// TIA Portal V17 program export: 1 tag tables, 0 data types, 1 data blocks, 2 code blocks (in call order from the OBs), 5 instance data blocks

VAR_GLOBAL   // PLC tag table "Default tag table"
END_VAR

DATA_BLOCK "IO"   // DB1
{ S7_Optimized_Access := 'TRUE' }
VERSION : 0.1
// stored: AutoNumber true, IsOnlyStoredInLoadMemory false, IsRetainMemResEnabled false, IsWriteProtectedInAS false, MemoryReserve 100
   VAR
      start : Bool;
      stop : Bool := true;
      awaryjeOproznianie : Bool := true;
      czasParzenia : Time := T#5S;
      zadanaIloscWody : Real := 500.0;
      zadanaIloscHerbaty : Real := 15.0;
      temperatura : Int;
      przenosnikM1 : Bool;
      mieszalnikM2 : Bool;
      podgrzewaczG1 : Bool;
      otworzZaworZ1 : Bool;
      otworzZasuweZ2 : Bool;
      otworzZasuweZ3 : Bool;
      wodaPoziom : Real;
      lisciePoziom : Real;
      glownyPoziom : Real;
   END_VAR
BEGIN
END_DATA_BLOCK

ORGANIZATION_BLOCK "Main"   // OB1, LAD, ProgramCycle
TITLE = "Main Program Sweep (Cycle)"
{ S7_Optimized_Access := 'TRUE' }
VERSION : 0.1
// stored: AutoNumber true, IsIECCheckEnabled false, SetENOAutomatically false
   VAR_INPUT
      Initial_Call : Bool;   // Initial call of this OB
      Remanence : Bool;   // =True, if remanent data are available
   END_VAR
BEGIN

REGION Network 1: Zadanie finałowe kategorii EKSPERT
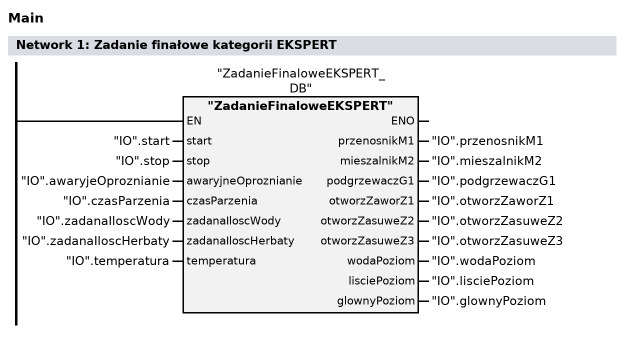
   RUNG wire#powerrail
      "ZadanieFinaloweEKSPERT_DB"(start := "IO".start, stop := "IO".stop, awaryjneOproznianie := "IO".awaryjeOproznianie, czasParzenia := "IO".czasParzenia, zadanaIloscWody := "IO".zadanaIloscWody, zadanaIloscHerbaty := "IO".zadanaIloscHerbaty, temperatura := "IO".temperatura, przenosnikM1 => "IO".przenosnikM1, mieszalnikM2 => "IO".mieszalnikM2, podgrzewaczG1 => "IO".podgrzewaczG1, otworzZaworZ1 => "IO".otworzZaworZ1, otworzZasuweZ2 => "IO".otworzZasuweZ2, otworzZasuweZ3 => "IO".otworzZasuweZ3, wodaPoziom => "IO".wodaPoziom, lisciePoziom => "IO".lisciePoziom, glownyPoziom => "IO".glownyPoziom)
   END_RUNG
   // the same network as SCL:
   "ZadanieFinaloweEKSPERT_DB"(start := "IO".start,   // "ZadanieFinaloweEKSPERT"
                           stop := "IO".stop,
                           awaryjneOproznianie := "IO".awaryjeOproznianie,
                           czasParzenia := "IO".czasParzenia,
                           zadanaIloscWody := "IO".zadanaIloscWody,
                           zadanaIloscHerbaty := "IO".zadanaIloscHerbaty,
                           temperatura := "IO".temperatura,
                           przenosnikM1 => "IO".przenosnikM1,
                           mieszalnikM2 => "IO".mieszalnikM2,
                           podgrzewaczG1 => "IO".podgrzewaczG1,
                           otworzZaworZ1 => "IO".otworzZaworZ1,
                           otworzZasuweZ2 => "IO".otworzZasuweZ2,
                           otworzZasuweZ3 => "IO".otworzZasuweZ3,
                           wodaPoziom => "IO".wodaPoziom,
                           lisciePoziom => "IO".lisciePoziom,
                           glownyPoziom => "IO".glownyPoziom);
END_REGION
END_ORGANIZATION_BLOCK

FUNCTION_BLOCK "ZadanieFinaloweEKSPERT"   // FB1, LAD
TITLE = Zadanie finałowe kategorii EKSPERT
{ S7_Optimized_Access := 'TRUE' }
VERSION : 0.1
// stored: AutoNumber true, IsIECCheckEnabled false, IsRetainMemResEnabled false, MemoryReserve 100, SetENOAutomatically false, UDAEnableTagReadback false
   VAR_INPUT
      start : Bool;
      stop : Bool;
      awaryjneOproznianie : Bool;
      czasParzenia : Time;
      zadanaIloscWody : Real;
      zadanaIloscHerbaty : Real;
      temperatura : Int;
   END_VAR
   VAR_OUTPUT
      przenosnikM1 : Bool;
      mieszalnikM2 : Bool;
      podgrzewaczG1 : Bool;
      otworzZaworZ1 : Bool;
      otworzZasuweZ2 : Bool;
      otworzZasuweZ3 : Bool;
      wodaPoziom : Real := 10000.0;
      lisciePoziom : Real := 100.0;
      glownyPoziom : Real;
   END_VAR
   VAR
      S1 : Bool;
      S2 : Bool;
      S3 : Bool;
      S4 : Bool;
      S5 : Bool;
      S0 : Bool;
      start_edge : Bool;
      stop_edge : Bool;
      awaryjne_edge : Bool;
      S1_Clock : Bool;
      w_glownym_wody : Real;
      w_glownym_herbaty : Real;
      S3_clock : Bool;
      M2_edge : Bool;
      S5_clock : Bool;
   END_VAR
   VAR_TEMP
      temp_norm : Real;
      tempC : Real;
   END_VAR
   VAR_TEMP   // added for the SCL form of the ladder/FBD networks
      _w1 : Bool;
      _w2 : Bool;
      _w3 : Bool;
   END_VAR
BEGIN

REGION Network 1
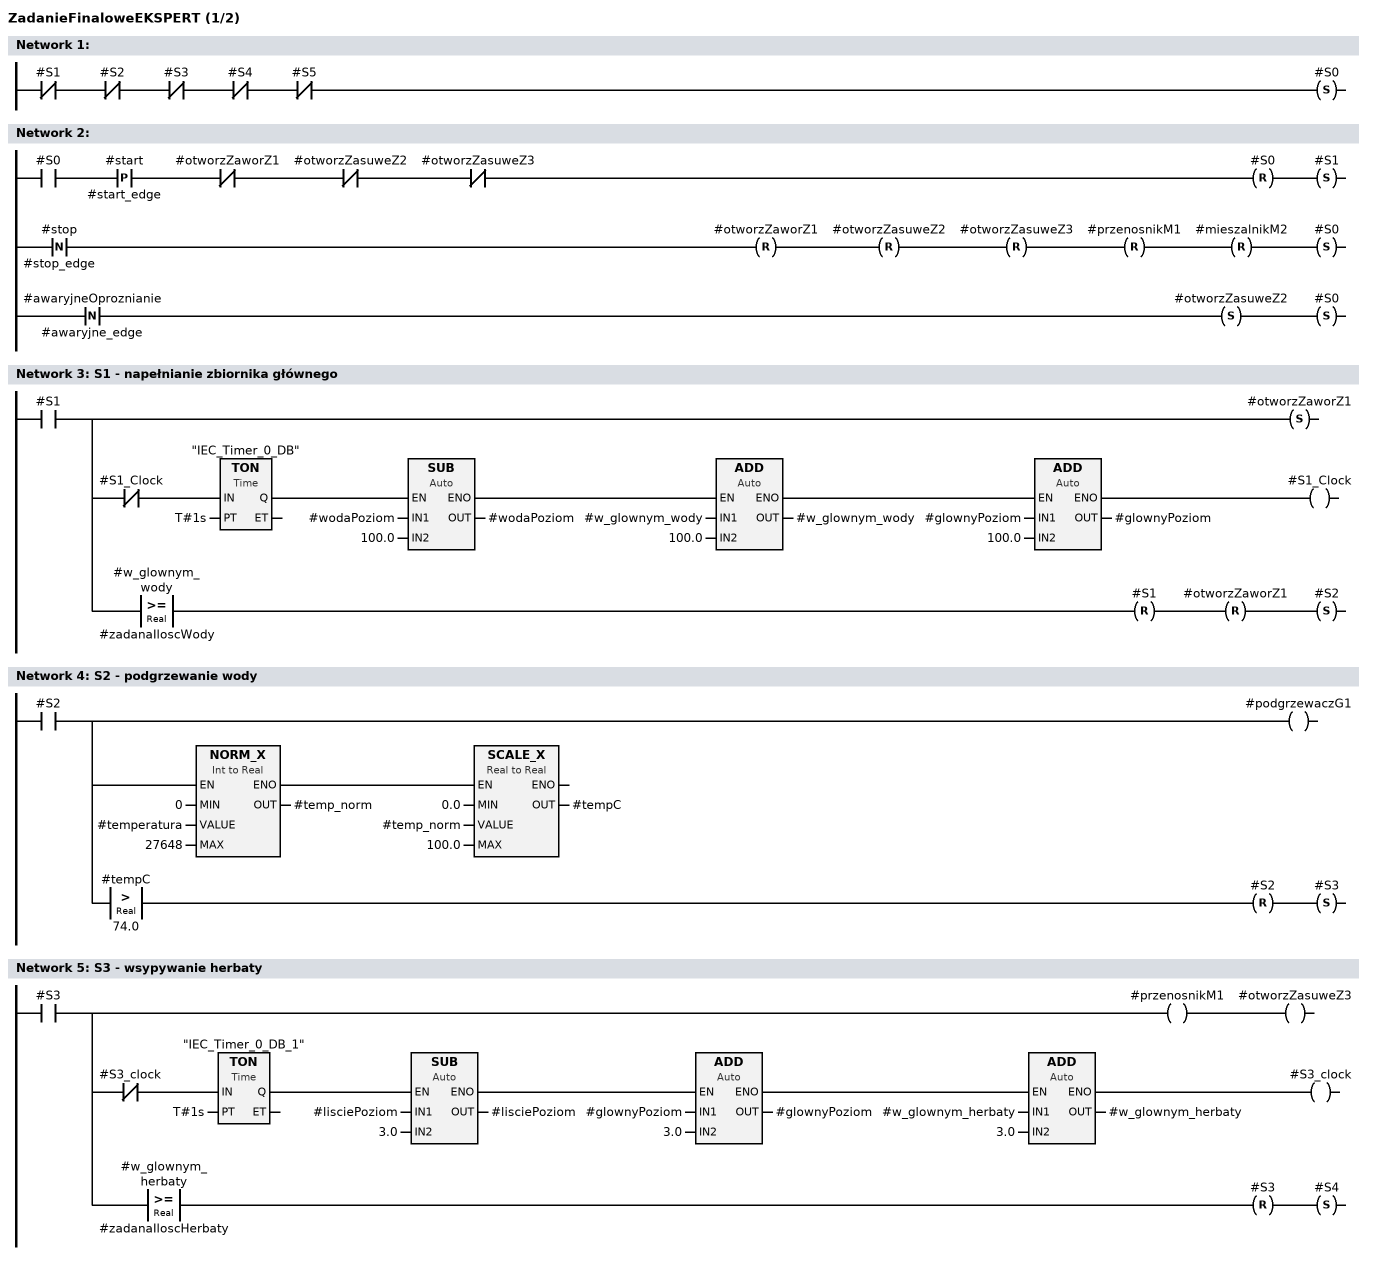
   RUNG wire#powerrail
      I_Contact( #S1 )
      I_Contact( #S2 )
      I_Contact( #S3 )
      I_Contact( #S4 )
      I_Contact( #S5 )
      S_Coil( #S0 )
   END_RUNG
   // the same network as SCL:
   IF NOT #S1 AND NOT #S2 AND NOT #S3 AND NOT #S4 AND NOT #S5 THEN #S0 := TRUE; END_IF;
END_REGION

REGION Network 2
   RUNG wire#powerrail
      Contact( #S0 )
      P_Contact(operand := #start, bit := #start_edge)
      I_Contact( #otworzZaworZ1 )
      I_Contact( #otworzZasuweZ2 )
      I_Contact( #otworzZasuweZ3 )
      R_Coil( #S0 )
      S_Coil( #S1 )
   END_RUNG
   RUNG wire#powerrail
      N_Contact(operand := #stop, bit := #stop_edge)
      R_Coil( #otworzZaworZ1 )
      R_Coil( #otworzZasuweZ2 )
      R_Coil( #otworzZasuweZ3 )
      R_Coil( #przenosnikM1 )
      R_Coil( #mieszalnikM2 )
      S_Coil( #S0 )
   END_RUNG
   RUNG wire#powerrail
      N_Contact(operand := #awaryjneOproznianie, bit := #awaryjne_edge)
      S_Coil( #otworzZasuweZ2 )
      S_Coil( #S0 )
   END_RUNG
   // the same network as SCL:
   #_w1 := #S0 AND #start AND NOT #start_edge;   // rising edge of #start
   #start_edge := #start;
   IF #_w1 AND NOT #otworzZaworZ1 AND NOT #otworzZasuweZ2 AND NOT #otworzZasuweZ3 THEN
       #S0 := FALSE;
       #S1 := TRUE;
   END_IF;
   #_w2 := NOT #stop AND #stop_edge;   // falling edge of #stop
   #stop_edge := #stop;
   IF #_w2 THEN
       #otworzZaworZ1 := FALSE;
       #otworzZasuweZ2 := FALSE;
       #otworzZasuweZ3 := FALSE;
       #przenosnikM1 := FALSE;
       #mieszalnikM2 := FALSE;
       #S0 := TRUE;
   END_IF;
   #_w3 := NOT #awaryjneOproznianie AND #awaryjne_edge;   // falling edge of #awaryjneOproznianie
   #awaryjne_edge := #awaryjneOproznianie;
   IF #_w3 THEN
       #otworzZasuweZ2 := TRUE;
       #S0 := TRUE;
   END_IF;
END_REGION

REGION Network 3: S1 - napełnianie zbiornika głównego
   RUNG wire#powerrail
      Contact( #S1 )
      wire#w1
      S_Coil( #otworzZaworZ1 )
   END_RUNG
   RUNG wire#w1
      I_Contact( #S1_Clock )
      { S7_Templates := "time_type := Time" } "IEC_Timer_0_DB".TON(pt := T#1s, et =>)
      Sub(in1 := #wodaPoziom, in2 := 100.0, out => #wodaPoziom)
      Add(in1 := #w_glownym_wody, in2 := 100.0, out => #w_glownym_wody)
      Add(in1 := #glownyPoziom, in2 := 100.0, out => #glownyPoziom)
      Coil( #S1_Clock )
   END_RUNG
   RUNG wire#w1
      { S7_Templates := "SrcType := Real" } GE_Contact(in1 := #w_glownym_wody, in2 := #zadanaIloscWody)
      R_Coil( #S1 )
      R_Coil( #otworzZaworZ1 )
      S_Coil( #S2 )
   END_RUNG
   // the same network as SCL:
   IF #S1 THEN #otworzZaworZ1 := TRUE; END_IF;
   "IEC_Timer_0_DB".TON(IN := #S1 AND NOT #S1_Clock, PT := T#1s);
   IF "IEC_Timer_0_DB".Q THEN
       #wodaPoziom := #wodaPoziom - 100.0;
       #w_glownym_wody := #w_glownym_wody + 100.0;
       #glownyPoziom := #glownyPoziom + 100.0;
   END_IF;
   #S1_Clock := "IEC_Timer_0_DB".Q;
   #_w1 := #S1 AND (#w_glownym_wody >= #zadanaIloscWody);
   IF #_w1 THEN
       #S1 := FALSE;
       #otworzZaworZ1 := FALSE;
       #S2 := TRUE;
   END_IF;
END_REGION

REGION Network 4: S2 - podgrzewanie wody
   RUNG wire#powerrail
      Contact( #S2 )
      wire#w1
      Coil( #podgrzewaczG1 )
   END_RUNG
   RUNG wire#w1
      { S7_Templates := "[SrcType := Int, DestType := Real]" } Normalize(min := 0, value := #temperatura, max := 27648, out => #temp_norm)
      { S7_Templates := "[SrcType := Real, DestType := Real]" } Scale(min := 0.0, value := #temp_norm, max := 100.0, out => #tempC)
   END_RUNG
   RUNG wire#w1
      { S7_Templates := "SrcType := Real" } GT_Contact(in1 := #tempC, in2 := 74.0)
      R_Coil( #S2 )
      S_Coil( #S3 )
   END_RUNG
   // the same network as SCL:
   #podgrzewaczG1 := #S2;
   IF #S2 THEN
       #temp_norm := NORM_X(MIN := 0, VALUE := #temperatura, MAX := 27648);
       #tempC := SCALE_X(MIN := 0.0, VALUE := #temp_norm, MAX := 100.0);
   END_IF;
   #_w1 := #S2 AND (#tempC > 74.0);
   IF #_w1 THEN
       #S2 := FALSE;
       #S3 := TRUE;
   END_IF;
END_REGION

REGION Network 5: S3 - wsypywanie herbaty
   RUNG wire#powerrail
      Contact( #S3 )
      wire#w1
      Coil( #przenosnikM1 )
      Coil( #otworzZasuweZ3 )
   END_RUNG
   RUNG wire#w1
      I_Contact( #S3_clock )
      { S7_Templates := "time_type := Time" } "IEC_Timer_0_DB_1".TON(pt := T#1s, et =>)
      Sub(in1 := #lisciePoziom, in2 := 3.0, out => #lisciePoziom)
      Add(in1 := #glownyPoziom, in2 := 3.0, out => #glownyPoziom)
      Add(in1 := #w_glownym_herbaty, in2 := 3.0, out => #w_glownym_herbaty)
      Coil( #S3_clock )
   END_RUNG
   RUNG wire#w1
      { S7_Templates := "SrcType := Real" } GE_Contact(in1 := #w_glownym_herbaty, in2 := #zadanaIloscHerbaty)
      R_Coil( #S3 )
      S_Coil( #S4 )
   END_RUNG
   // the same network as SCL:
   #przenosnikM1 := #S3;
   #otworzZasuweZ3 := #S3;
   "IEC_Timer_0_DB_1".TON(IN := #S3 AND NOT #S3_clock, PT := T#1s);
   IF "IEC_Timer_0_DB_1".Q THEN
       #lisciePoziom := #lisciePoziom - 3.0;
       #glownyPoziom := #glownyPoziom + 3.0;
       #w_glownym_herbaty := #w_glownym_herbaty + 3.0;
   END_IF;
   #S3_clock := "IEC_Timer_0_DB_1".Q;
   #_w1 := #S3 AND (#w_glownym_herbaty >= #zadanaIloscHerbaty);
   IF #_w1 THEN
       #S3 := FALSE;
       #S4 := TRUE;
   END_IF;
END_REGION

REGION Network 6: S4 - mieszanie
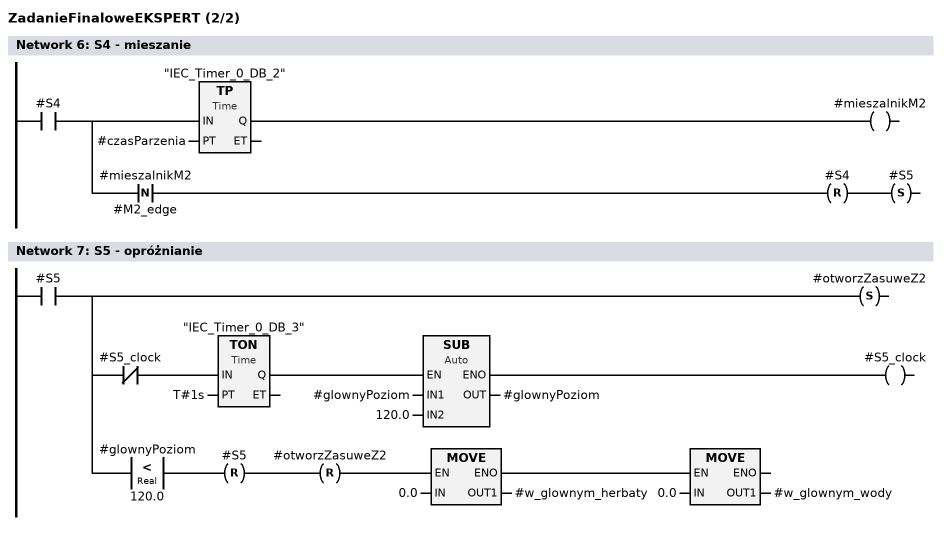
   RUNG wire#powerrail
      Contact( #S4 )
      wire#w1
      { S7_Templates := "time_type := Time" } "IEC_Timer_0_DB_2".TP(pt := #czasParzenia, et =>)
      Coil( #mieszalnikM2 )
   END_RUNG
   RUNG wire#w1
      N_Contact(operand := #mieszalnikM2, bit := #M2_edge)
      R_Coil( #S4 )
      S_Coil( #S5 )
   END_RUNG
   // the same network as SCL:
   "IEC_Timer_0_DB_2".TP(IN := #S4, PT := #czasParzenia);
   #mieszalnikM2 := "IEC_Timer_0_DB_2".Q;
   #_w1 := #S4 AND NOT #mieszalnikM2 AND #M2_edge;   // falling edge of #mieszalnikM2
   #M2_edge := #mieszalnikM2;
   IF #_w1 THEN
       #S4 := FALSE;
       #S5 := TRUE;
   END_IF;
END_REGION

REGION Network 7: S5 - opróżnianie
   RUNG wire#powerrail
      Contact( #S5 )
      wire#w1
      S_Coil( #otworzZasuweZ2 )
   END_RUNG
   RUNG wire#w1
      I_Contact( #S5_clock )
      { S7_Templates := "time_type := Time" } "IEC_Timer_0_DB_3".TON(pt := T#1s, et =>)
      Sub(in1 := #glownyPoziom, in2 := 120.0, out => #glownyPoziom)
      Coil( #S5_clock )
   END_RUNG
   RUNG wire#w1
      { S7_Templates := "SrcType := Real" } LT_Contact(in1 := #glownyPoziom, in2 := 120.0)
      R_Coil( #S5 )
      R_Coil( #otworzZasuweZ2 )
      Move(in := 0.0, out1 => #w_glownym_herbaty)
      Move(in := 0.0, out1 => #w_glownym_wody)
   END_RUNG
   // the same network as SCL:
   IF #S5 THEN #otworzZasuweZ2 := TRUE; END_IF;
   "IEC_Timer_0_DB_3".TON(IN := #S5 AND NOT #S5_clock, PT := T#1s);
   IF "IEC_Timer_0_DB_3".Q THEN #glownyPoziom := #glownyPoziom - 120.0; END_IF;
   #S5_clock := "IEC_Timer_0_DB_3".Q;
   #_w1 := #S5 AND (#glownyPoziom < 120.0);
   IF #_w1 THEN
       #S5 := FALSE;
       #otworzZasuweZ2 := FALSE;
       #w_glownym_herbaty := 0.0;
       #w_glownym_wody := 0.0;
   END_IF;
END_REGION
END_FUNCTION_BLOCK

DATA_BLOCK "ZadanieFinaloweEKSPERT_DB"   // DB2
VERSION : 0.1
// stored: AutoNumber true, InstanceOfName ZadanieFinaloweEKSPERT, InstanceOfType FB
"ZadanieFinaloweEKSPERT"
BEGIN
END_DATA_BLOCK

DATA_BLOCK "IEC_Timer_0_DB"   // DB3
{ S7_Optimized_Access := 'TRUE' }
// stored: AutoNumber true, InstanceOfName IEC_TIMER, OfSystemLibElement IEC_TIMER, OfSystemLibVersion 1.0
"IEC_TIMER"
   // VAR
   //    PT : Time;
   //    ET { ExternalWritable := 'False'} : Time;
   //    IN : Bool;
   //    Q { ExternalWritable := 'False'} : Bool;
   // END_VAR
BEGIN
END_DATA_BLOCK

DATA_BLOCK "IEC_Timer_0_DB_1"   // DB4
{ S7_Optimized_Access := 'TRUE' }
// stored: AutoNumber true, InstanceOfName IEC_TIMER, OfSystemLibElement IEC_TIMER, OfSystemLibVersion 1.0
"IEC_TIMER"
   // VAR
   //    PT : Time;
   //    ET { ExternalWritable := 'False'} : Time;
   //    IN : Bool;
   //    Q { ExternalWritable := 'False'} : Bool;
   // END_VAR
BEGIN
END_DATA_BLOCK

DATA_BLOCK "IEC_Timer_0_DB_2"   // DB5
{ S7_Optimized_Access := 'TRUE' }
// stored: AutoNumber true, InstanceOfName IEC_TIMER, OfSystemLibElement IEC_TIMER, OfSystemLibVersion 1.0
"IEC_TIMER"
   // VAR
   //    PT : Time;
   //    ET { ExternalWritable := 'False'} : Time;
   //    IN : Bool;
   //    Q { ExternalWritable := 'False'} : Bool;
   // END_VAR
BEGIN
END_DATA_BLOCK

DATA_BLOCK "IEC_Timer_0_DB_3"   // DB6
{ S7_Optimized_Access := 'TRUE' }
// stored: AutoNumber true, InstanceOfName IEC_TIMER, OfSystemLibElement IEC_TIMER, OfSystemLibVersion 1.0
"IEC_TIMER"
   // VAR
   //    PT : Time;
   //    ET { ExternalWritable := 'False'} : Time;
   //    IN : Bool;
   //    Q { ExternalWritable := 'False'} : Bool;
   // END_VAR
BEGIN
END_DATA_BLOCK
